{attribute 'enable_dynamic_creation'}
TYPE ST_SequenceInfo :
STRUCT
	nSequId 		: UDINT;			//4 Byte
	nStepNr 		: UINT;				//2 Byte
	eSequenceState	: E_SequenceState;	//1 Byte
	eStepState		: E_StepState;		//1 Byte
	nInfo			: DINT;				//4 Byte
END_STRUCT
END_TYPE

(* stored: Version 1.1.0.1, ProductVersion 3.1.4022.10
   DUT ST_SequenceInfo: Id {54a70cf3-1e23-43f3-b254-f3d4dd6e8f77} *)
